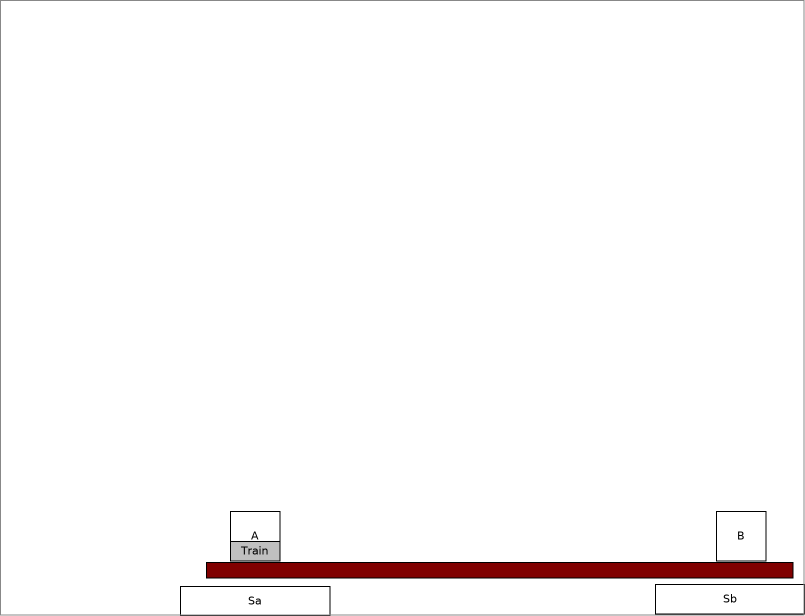
VISUALIZATION Visualization  // 805x616
    Rectangle (206,562 587x16)
    Rectangle (230,511 50x50), "A"
    Rectangle (716,511 50x50), "B"
    Rectangle (230,541 50x20), "Train"
        p3560616238: Motor_Control.Pos
    Rectangle (180,586 150x30), "Sa", colour toggle: GVL.qxA
    Rectangle (655,584 150x30), "Sb", colour toggle: GVL.qxB
END_VISUALIZATION

(* stored: Version 1.1.0.1, ProductVersion 3.1.4024.12
   Visu Visualization: Id {379103cc-b65c-4590-a6c5-e0a2146f16b5} *)
